GLOBALCONSTANTS DefaultPool_Dreieck_Bargraph (* Bargraph geometry and scale constants (Length, ScalePx, Min, Max, Type) *)
  PACKAGE Uebungen::const::UT::Dreieck;
  VAR_GLOBAL CONSTANT
    LinearBargraph_ScalePx : REAL := 1.0;
    LinearBargraph_LengthPx : REAL := 84.0;
    LinearBargraph_Min : REAL := 0.0;
    LinearBargraph_Max : REAL := 84.0;
    LinearBargraph_Type : USINT := 3;
  END_VAR
END_GLOBALCONSTANTS
